// Stage diagnostic buffer limits.
{attribute 'qualified_only'}
VAR_GLOBAL CONSTANT
	MAX_PANIC_MSG: UDINT(1..16#7FFFFFFF) := 10; // Panic buffer entries; do not set to 0.
	MAX_WARN_MSG: UDINT(1..16#7FFFFFFF) := 10; // Warning buffer entries; do not set to 0.
	VALIDATION_GUARD: UDINT(1..16#7FFFFFFF) := 100_000;
END_VAR

(* stored: Version 1.1.0.1
   GVL Param: Id {bc9b684f-96ba-4011-afc3-650f65d44b69}, ParameterList True *)
